(* CoDeSys 2.3 export: LENGTH.EXP *)

(* Data type in INT *)
TYPE Length : INT;
END_TYPE
